// TwinCAT 3 PLC project PLC
// ProgramVersion: 3.1.4026.24
// libraries:
//   PS_DcUpsEC, * (Phoenix Contact GmbH & Co.KG)
//   Tc2_Standard, * (Beckhoff Automation GmbH)
//   Tc2_System, * (Beckhoff Automation GmbH)
// project tree:
//   / PlcTask.TcTTO
//   POUs/ MAIN.TcPOU
// real-time tasks:
//   TASK PlcTask: cycle T#10ms, priority 20, ADS port 350
// I/O:
//   DEVICE Device 3 (EtherCAT), AmsNetId 5.176.90.10.4.1
//     Term 1 (EK1200) [EK1200-5000 EtherCAT Power supply (2A E-Bus)]
//       Term 5 (EK1122) [EK1122 2 port EtherCAT junction]
//         Box 1 (Uninterruptible Power Supply) [QUINT4-UPS/24DC/24DC/10/EC]
// variable links:
//   PLC/PLC Instance <-> Device 3 (EtherCAT)/Term 1 (EK1200)/Term 5 (EK1122)/Box 1 (Uninterruptible Power Supply)
//     PlcTask Inputs/MAIN.arrInputPD @bit {304..432 step 32} <-> TxPDO 1/BATTERY {1..5} ALARMS  (5 links)
//     PlcTask Inputs/MAIN.arrInputPD @bit 80 <-> TxPDO 1/STATUS ACTUAL INPUT CURRENT
//     PlcTask Inputs/MAIN.arrInputPD @bit 64 <-> TxPDO 1/STATUS ACTUAL INPUT VOLTAGE
//     PlcTask Inputs/MAIN.arrInputPD @bit 112 <-> TxPDO 1/STATUS ACTUAL OUTPUT CURRENT 1
//     PlcTask Inputs/MAIN.arrInputPD @bit 96 <-> TxPDO 1/STATUS ACTUAL OUTPUT VOLTAGE 1
//     PlcTask Inputs/MAIN.arrInputPD @bit 128 <-> TxPDO 1/STATUS BATTERY ACTUAL VOLTAGE
//     PlcTask Inputs/MAIN.arrInputPD @bit 144 <-> TxPDO 1/STATUS BATTERY CHARGE CURRENT
//     PlcTask Inputs/MAIN.arrInputPD @bit 160 <-> TxPDO 1/STATUS BATTERY TEMPERATURE
//     PlcTask Inputs/MAIN.arrInputPD @bit 176 <-> TxPDO 1/STATUS DEVICE TEMPERATURE
//     PlcTask Inputs/MAIN.arrInputPD <-> TxPDO 1/STATUS FUNCTIONS
//     PlcTask Inputs/MAIN.arrInputPD @bit 32 <-> TxPDO 1/STATUS INTERFACE
//     PlcTask Inputs/MAIN.arrInputPD @bit 192 <-> TxPDO 1/STATUS SOC REMAINING TIME
//     PlcTask Inputs/MAIN.arrInputPD @bit 224 <-> TxPDO 1/STATUS SOC REMAINING TIME PC SHUTDOWN
//     PlcTask Inputs/MAIN.arrInputPD @bit 240 <-> TxPDO 1/STATUS SOH REMAINING LIFETIME
//     PlcTask Inputs/MAIN.arrInputPD @bit 272 <-> TxPDO 1/UPS DIAGNOSIS ALARMS
//     PlcTask Inputs/MAIN.arrInputPD @bit 256 <-> TxPDO 1/UPS PROCESS ALARMS

CONFIGURATION PLC
    RESOURCE PLC ON TwinCAT3
        TASK PlcTask(INTERVAL := T#10ms, PRIORITY := 20);
        PROGRAM MAIN WITH PlcTask : MAIN;
    END_RESOURCE
END_CONFIGURATION

// ---- POUs/MAIN.TcPOU
PROGRAM MAIN
VAR
	USVCyclicComm : PS_Q4_DcUpsEC_Cyclic_3;
	USVParamComm  : PS_Q4_DcUpsEC_Param_1;
	
	arrInputPD	AT%I* : ARRAY [0..30] OF WORD;	// Connect Multilink of TxPDO here
	
END_VAR

USVCyclicComm(xActivate:=TRUE,arrInputPD:=arrInputPD);
// USVParamComm();

END_PROGRAM
